// TwinCAT 3 PLC project RoboConnect_Tests
// Title: RoboConnect.Tests
// Company: RoboConnect
// Author: RoboConnect_Maintainer
// ProjectVersion: 0.0.5.0
// Description: 0.1.0.0 Branding update 0.0.5.0 cleans up project 0.0.0.4 updates to new tcrobot 0.0.0.3 Remove tcrobot instances from tests 0.0.0.2 Adds IO tests 0.0.0.1 Adds connection tests
// ProgramVersion: 3.1.4024.0
// libraries:
//   Intecre.Utilities, * (Intecre Ltd)
//   RoboConnect, * (RoboConnect)
//   Tc2_Standard, * (Beckhoff Automation GmbH)
//   tcl_SimpleUnitTestLibrary, * (Red Rock Controls Limited)
// project tree:
//   Code/Mocks/ T_MockBoolCommandTask.TcPOU, T_MockCommandTask.TcPOU, T_MockNumberCommandTask.TcPOU, T_MockTcRobot.TcPOU
//   Code/RoboConnect/Admin Tests/Disable/ T_RoboConnect_Disable_DisabledTrue.TcPOU
//   Code/RoboConnect/Admin Tests/Enable/ T_RoboConnect_Enable_RobotEnabled.TcPOU
//   Code/RoboConnect/ConnectionTests/ T_RoboConnect_WhenCalledWithLowTimeout_FailsConnection.TcPOU, T_RoboConnect_WhenCalled_IsConnectedTrue.TcPOU
//   Code/RoboConnect/IO Tests/AnalogOutput/ T_TcRobot_GetAnalogOutput_CorrectIndexPasses.TcPOU, T_TcRobot_SetAnalogOutput_IncorrectIndexFails.TcPOU, T_TcRobot_SetAnalogOutput_CorrectIndexPasses.TcPOU, T_TcRobot_GetAnalogOutput_IncorrectIndexFails.TcPOU, T_TcRobot_SetAnalogOutput_TimeoutFails.TcPOU
//   Code/RoboConnect/IO Tests/DigitalOutput/ T_TcRobot_SetDigitalOutputTimeout_Fails.TcPOU, T_TcRobot_GetDigitalOutput_CorrectIndexPasses.TcPOU, T_TcRobot_SetDigitalOutput_IncorrectIndexFails.TcPOU, T_TcRobot_SetDigitalOutput_CorrectIndexPasses.TcPOU, T_TcRobot_GetDigitalOutput_ReturnsTrueOutput.TcPOU, T_TcRobot_GetDigitalOutput_IncorrectIndexFails.TcPOU
//   Code/RoboConnect/IO Tests/ToolAnalogOutput/ T_TcRobot_GetToolAnalogOutput_CorrectIndexPasses.TcPOU, T_TcRobot_SetToolAnalogOutput_TimeoutFails.TcPOU, T_TcRobot_SetToolAnalogOutput_IncorrectIndexFails.TcPOU, T_TcRobot_SetToolAnalogOutput_CorrectIndexPasses.TcPOU, T_TcRobot_GetToolAnalogOutput_IncorrectIndexFails.TcPOU
//   Code/RoboConnect/IO Tests/ToolDigitalOutput/ T_TcRobot_SetToolDigitalOutputTimeout_Fails.TcPOU, T_TcRobot_GetToolDigitalOutput_CorrectIndexPasses.TcPOU, T_TcRobot_SetToolDigitalOutput_IncorrectIndexFails.TcPOU, T_TcRobot_SetToolDigitalOutput_CorrectIndexPasses.TcPOU, T_TcRobot_GetToolDigitalOutput_IncorrectIndexFails.TcPOU, T_TcRobot_SetToolDigitalOutput_ReturnsTrueOutput.TcPOU
//   Code/RoboConnect/ T_TcRobot_DisableNotConnected_ReturnsFalse.TcPOU, T_TcRobot_MoveJWrongCount_ReturnsFalse.TcPOU
// (motion and I/O tree: see PLC project roboconnect)
// real-time tasks:
//   TASK PlcTask: cycle T#10ms, priority 22, ADS port 350
//   TASK PlcTask1: cycle T#10ms, priority 21, ADS port 351

// ---- Code/Mocks/T_MockBoolCommandTask.TcPOU
FUNCTION_BLOCK T_MockBoolCommandTask IMPLEMENTS I_BoolResultTask
VAR_INPUT
  _Busy, _Done, _Error, _Timeout : BOOL;
  _Result : BOOL;
END_VAR

METHOD Abort
END_METHOD

PROPERTY Available : BOOL
GET
END_GET
END_PROPERTY

PROPERTY Busy : BOOL
GET
Busy := _busy;
END_GET
END_PROPERTY

METHOD CyclicLogic
END_METHOD

PROPERTY Done : BOOL
GET
Done := _Done;
END_GET
END_PROPERTY

PROPERTY Error : BOOL
GET
Error := _Error;
END_GET
END_PROPERTY

PROPERTY ErrorId : STRING
GET
END_GET
END_PROPERTY

METHOD Execute : BOOL
END_METHOD

METHOD Free
END_METHOD

PROPERTY Result : BOOL
GET
Result := _Result;
END_GET
END_PROPERTY

PROPERTY Timeout : BOOL
GET
Timeout := _Timeout;
END_GET
END_PROPERTY

END_FUNCTION_BLOCK

// ---- Code/Mocks/T_MockCommandTask.TcPOU
FUNCTION_BLOCK T_MockCommandTask IMPLEMENTS I_Task
VAR_INPUT
  _Busy, _Done, _Error, _Timeout : BOOL;
  _Result : LREAL;
END_VAR

METHOD Abort
END_METHOD

PROPERTY Available : BOOL
GET
END_GET
END_PROPERTY

PROPERTY Busy : BOOL
GET
Busy := _Busy;
END_GET
END_PROPERTY

METHOD CyclicLogic
END_METHOD

PROPERTY Done : BOOL
GET
Done := _Done;
END_GET
END_PROPERTY

PROPERTY Error : BOOL
GET
Error := _Error;
END_GET
END_PROPERTY

PROPERTY ErrorId : STRING
GET
END_GET
END_PROPERTY

METHOD Execute : BOOL
END_METHOD

METHOD Free
END_METHOD

PROPERTY Timeout : BOOL
GET
Timeout := _Timeout;
END_GET
END_PROPERTY

END_FUNCTION_BLOCK

// ---- Code/Mocks/T_MockNumberCommandTask.TcPOU
FUNCTION_BLOCK T_MockNumberCommandTask IMPLEMENTS I_NumberResultTask
VAR_INPUT
  _Busy, _Done, _Error, _Timeout : BOOL;
  _Result : LREAL;
END_VAR

METHOD Abort
END_METHOD

PROPERTY Available : BOOL
GET
END_GET
END_PROPERTY

PROPERTY Busy : BOOL
GET
Busy := _Busy;
END_GET
END_PROPERTY

METHOD CyclicLogic
END_METHOD

PROPERTY Done : BOOL
GET
Done := _Done;
END_GET
END_PROPERTY

PROPERTY Error : BOOL
GET
Error := _Error;
END_GET
END_PROPERTY

PROPERTY ErrorId : STRING
GET
END_GET
END_PROPERTY

METHOD Execute : BOOL
END_METHOD

METHOD Free
END_METHOD

PROPERTY Result : LREAL
GET
Result := _Result;
END_GET
END_PROPERTY

PROPERTY Timeout : BOOL
GET
Timeout := _Timeout;
END_GET
END_PROPERTY

END_FUNCTION_BLOCK

// ---- Code/Mocks/T_MockTcRobot.TcPOU
FUNCTION_BLOCK T_MockRoboConnect IMPLEMENTS I_RoboConnect
VAR_INPUT
  _error, _isBusy, _isDone, _isEnabled : BOOL;
  _errorId : UINT;
  _axisCount : UINT;
  _position, _toolPosition : ST_CartesianPoint;
END_VAR
VAR
  state, prevState : (INIT,
    IDLE,
    READY,
    ERROR_STATE) := INIT;

  initalised : BOOL;
  connectionTimer : TON;
  tasktimer : TON;
  _connection : I_Connection;
  _commandQueue : I_CommandQueue;
  _commandTask : T_MockCommandTask;
  _boolCommandTask : T_MockBoolCommandTask;
  _numberCommandTask : T_MockNumberCommandTask;

  digitalOutputs : ARRAY[1..DIGITAL_OUTPUT_COUNT] OF BOOL;
  digitalIntputs : ARRAY[1..DIGITAL_INPUT_COUNT] OF BOOL;
  analogOutputs : ARRAY[1..ANALOG_OUTPUT_COUNT] OF LREAL;
  analogIntputs : ARRAY[1..ANALOG_INPUT_COUNT] OF LREAL;

  toolDigitalOutputs : ARRAY[1..TOOL_DIGITAL_OUTPUT] OF BOOL;
  toolDigitalIntputs : ARRAY[1..TOOL_DIGITAL_INPUT] OF BOOL;
  toolAnalogOutputs : ARRAY[1..TOOL_ANALOG_INPUT] OF LREAL;
  toolAnalogIntputs : ARRAY[1..TOOL_ANALOG_OUTPUT] OF LREAL;

  axes : ARRAY[1..AXIS_COUNT] OF LREAL;

END_VAR
VAR CONSTANT
  DIGITAL_OUTPUT_COUNT : UINT := 6;
  DIGITAL_INPUT_COUNT : UINT := 6;
  ANALOG_INPUT_COUNT : UINT := 6;
  ANALOG_OUTPUT_COUNT : UINT := 6;
  TOOL_ANALOG_OUTPUT : UINT := 2;
  TOOL_DIGITAL_OUTPUT : UINT := 2;
  TOOL_ANALOG_INPUT : UINT := 2;
  TOOL_DIGITAL_INPUT : UINT := 2;
  AXIS_COUNT : UINT := 6;

END_VAR

PROPERTY Busy : BOOL
GET
END_GET
END_PROPERTY

PROPERTY CartesianPosition : TcRobot.ST_CartesianPoint
GET
END_GET
END_PROPERTY

METHOD ClearError : BOOL
VAR_OUTPUT
	task	: TcRobot.I_Task;
END_VAR
END_METHOD

METHOD Connect : BOOL
connectionTimer( IN := FALSE );
connectionTimer( IN := TRUE );
END_METHOD

PROPERTY Connected : BOOL
GET
Connected := connectionTimer.Q;
END_GET
END_PROPERTY

METHOD CyclicLogic
connectionTimer();
taskTimer();

IF taskTimer.Q THEN
  _commandTask(_Timeout := TRUE);
END_IF
END_METHOD

METHOD Disable : BOOL
VAR_OUTPUT
  task : I_Task;
END_VAR
VAR
  resultTask : T_CommandTask;
END_VAR
IF NOT connectionTimer.Q THEN
  task := resultTask;
  RETURN;
END_IF
END_METHOD

METHOD Disconnect : BOOL
VAR_OUTPUT
  task : I_Task;
END_VAR
connectionTimer( IN := FALSE );
END_METHOD

PROPERTY Done : BOOL
GET
END_GET
END_PROPERTY

METHOD Enable : BOOL
VAR_OUTPUT
  task : I_Task;
END_VAR
END_METHOD

PROPERTY Enabled : BOOL
GET
END_GET
END_PROPERTY

PROPERTY Error : BOOL
GET
END_GET
END_PROPERTY

PROPERTY ErrorID : LREAL
GET
END_GET
END_PROPERTY

METHOD GetAnalogOutput : BOOL
VAR_INPUT
  Index : UINT;
END_VAR
VAR_OUTPUT
  task : I_NumberResultTask;
END_VAR
IF Index < 1 OR index > ANALOG_OUTPUT_COUNT THEN
  GetAnalogOutput := FALSE;
  RETURN;
END_IF

_commandTask(_Result := analogOutputs[Index]);
task := _numberCommandTask;

GetAnalogOutput := TRUE;
END_METHOD

METHOD GetAxisCurrents : BOOL
VAR_IN_OUT
  Values : ARRAY[*] OF LREAL;
END_VAR
VAR_OUTPUT
  task : I_Task;
END_VAR
END_METHOD

METHOD GetAxisPositions : BOOL
VAR_IN_OUT
  Values : ARRAY[*] OF LREAL;
END_VAR
VAR_OUTPUT
  task : I_Task;
END_VAR
END_METHOD

METHOD GetAxisTemperatures : BOOL
VAR_IN_OUT
  Values : ARRAY[*] OF LREAL;
END_VAR
VAR_OUTPUT
  task : I_Task;
END_VAR
END_METHOD

METHOD GetDigitalOutput : BOOL
VAR_INPUT
    Index : UINT;
END_VAR
VAR_OUTPUT
  task : I_BoolResultTask;
  value : BOOL;
END_VAR
VAR
  cmdTask : T_CommandTask;
END_VAR
IF Index < 1 OR index > DIGITAL_OUTPUT_COUNT THEN
  GetDigitalOutput := FALSE;
  RETURN;
END_IF

_commandTask(_Result := TO_LREAL(digitalOutputs[Index]), _Done := TRUE);
task := _boolCommandTask;

GetDigitalOutput := TRUE;
END_METHOD

METHOD GetJointPositions : BOOL (* false if incompatible array length*)
VAR_IN_OUT
	(* values overwritten with joint positions.*)
	  joints : ARRAY[*] OF LREAL;
END_VAR
END_METHOD

METHOD GetToolAnalogOutput : BOOL
VAR_INPUT
    Index : UINT;
END_VAR
VAR_OUTPUT
  task : I_NumberResultTask;
END_VAR
IF Index < 1 OR index > DIGITAL_OUTPUT_COUNT THEN
  GetToolAnalogOutput := FALSE;
  RETURN;
END_IF

_commandTask(_Result := toolAnalogOutputs[Index]);
task := _numberCommandTask;

GetToolAnalogOutput := TRUE;
END_METHOD

METHOD GetToolDigitalOutput : BOOL
VAR_INPUT
	Index	: UINT;
END_VAR
VAR_OUTPUT
	task	: I_BoolResultTask;
END_VAR
IF Index < 1 OR Index > TOOL_DIGITAL_OUTPUT THEN
  GetToolDigitalOutput := FALSE;
  RETURN;
END_IF

_commandTask(_Result := TO_LREAL(toolDigitalOutputs[Index]));
task := _boolCommandTask;

GetToolDigitalOutput := TRUE;
END_METHOD

METHOD Halt : BOOL
VAR_OUTPUT
  task : I_Task;
END_VAR
END_METHOD

METHOD IsAtCartesianPosition : BOOL
VAR_INPUT
	point	: TcRobot.ST_CartesianPoint;
END_VAR
END_METHOD

METHOD IsAtJointPosition : BOOL
VAR_IN_OUT
	(* positions 1..NumberOfAxes will be used. passed array should be dimensioned accordingly*)
  joints : ARRAY[*] OF LREAL; // positions 1..NumberOfAxes will be used. passed array should be dimensioned accordingly
END_VAR
END_METHOD

METHOD JogAxis : BOOL // default tool and user frame
VAR_INPUT
  axisIndex : UDINT; // joint or enumerated cartesian direction/vector. See concrete type docs for enumeration of cartesian coords.
  axisDirection : BOOL; // TRUE = positive, FALSE = negative
  jogType : E_JogType; // Cartesian or Joint space
END_VAR
VAR_OUTPUT
	task	: TcRobot.I_Task;
END_VAR
END_METHOD

METHOD JogAxisAdvanced : BOOL
VAR_INPUT
  axisIndex : UDINT; // joint or enumerated cartesian direction/vector. See concrete type docs for enumeration of cartesian coords.
  axisDirection : BOOL; // TRUE = positive, FALSE = negative
  jogType : E_JogType; // Cartesian or Joint space
  coordType : INT; // set to 0 to leave default
  user : INT; // set to 0 to leave default
  tool : INT; // set to 0 to leave default
END_VAR
VAR_OUTPUT
	task	: TcRobot.I_Task;
END_VAR
END_METHOD

PROPERTY Manufacturer : STRING
GET
END_GET
END_PROPERTY

PROPERTY Model : STRING
GET
END_GET
END_PROPERTY

METHOD MoveAbs : BOOL
VAR_INPUT
  point : ST_CartesianPoint;
END_VAR
VAR_OUTPUT
  task : I_Task;
END_VAR
END_METHOD

METHOD MoveJ : BOOL
VAR_IN_OUT
  joints : ARRAY[*] OF LREAL;
END_VAR
VAR_OUTPUT
  task : I_Task;
END_VAR
VAR
  returnedTask : T_CommandTask;
END_VAR
IF UPPER_BOUND(joints,1) > _axisCount THEN
  task := returnedTask;
  RETURN;
END_IF
END_METHOD

PROPERTY Position : ST_CartesianPoint
GET
END_GET
END_PROPERTY

METHOD Reset : BOOL
VAR_OUTPUT
  task : I_Task;
END_VAR
END_METHOD

PROPERTY Running : BOOL
GET
END_GET
END_PROPERTY

METHOD SetAnalogOutput : BOOL
VAR_INPUT
  Index : UINT;
  Value : LREAL;
END_VAR
VAR_OUTPUT
  task : I_Task;
END_VAR
IF Index < 1 OR index > DIGITAL_OUTPUT_COUNT THEN
  SetAnalogOutput := FALSE;
  RETURN;
END_IF

tasktimer.IN := FALSE;
tasktimer.IN := TRUE;

analogOutputs[Index] := Value;
task := _commandTask;

SetAnalogOutput := TRUE;
END_METHOD

METHOD SetAtPosDeltas : BOOL
VAR_INPUT
  atPosCartesianDeltas : ST_CartesianPoint;
END_VAR
VAR_IN_OUT
  atPosJointDeltas : ARRAY[*] OF LREAL; // positions 1..NumberOfAxes will be used. passed array should be dimensioned accordingly
END_VAR
END_METHOD

METHOD SetBufferMode : BOOL
VAR_INPUT
  BufferMode : E_BufferMode;
END_VAR
END_METHOD

METHOD SetCarteasianAcceleration : BOOL
VAR_INPUT
  Acceleration : LREAL;
END_VAR
VAR_OUTPUT
  task : I_Task;
END_VAR
END_METHOD

METHOD SetCartesianSpeed : BOOL
VAR_INPUT
  Speed : LREAL;
END_VAR
VAR_OUTPUT
  task : I_Task;
END_VAR
END_METHOD

METHOD PUBLIC SetConnectionTime  // set simulated connection time
VAR_INPUT
  connectionTime : TIME;
END_VAR
connectionTimer.PT := connectionTime;
END_METHOD

METHOD SetDigitalOutput : BOOL
VAR_INPUT
  Index : UINT;
  Value : BOOL;
END_VAR
VAR_OUTPUT
  task : I_Task;
END_VAR
IF Index < 1 OR index > DIGITAL_OUTPUT_COUNT THEN
  SetDigitalOutput := FALSE;
  RETURN;
END_IF

tasktimer.IN := FALSE;
tasktimer.IN := TRUE;

digitalOutputs[Index] := TRUE;
_commandTask(_Done := TRUE);
task := _commandTask;

SetDigitalOutput := TRUE;
END_METHOD

METHOD PUBLIC SetGeneralCommandResponseDuration : BOOL // This sets the duration that the task will take, used for causing timeout or done in the returned task
VAR_INPUT
    taskTime : TIME;
END_VAR
tasktimer.PT := taskTime;
END_METHOD

METHOD SetJogType : BOOL
VAR_INPUT
  JogType : E_JogType;
END_VAR
VAR_OUTPUT
  task : I_Task;
END_VAR
END_METHOD

METHOD SetJointAcceleration : BOOL
VAR_INPUT
  Acceleration : LREAL;
END_VAR
VAR_OUTPUT
  task : I_Task;
END_VAR
END_METHOD

METHOD SetJointSpeed : BOOL
VAR_INPUT
  Speed : LREAL;
END_VAR
VAR_OUTPUT
  task : I_Task;
END_VAR
END_METHOD

METHOD SetToolAnalogOutput : BOOL
VAR_INPUT
  Index : UINT;
  Value : LREAL;
END_VAR
VAR_OUTPUT
  task : I_Task;
END_VAR
IF Index > ANALOG_OUTPUT_COUNT THEN
  SetToolAnalogOutput := FALSE;
  RETURN;
END_IF

tasktimer.IN := FALSE;
tasktimer.IN := TRUE;

toolDigitalOutputs[Index] := TRUE;
task := _commandTask;

SetToolAnalogOutput := TRUE;
END_METHOD

METHOD SetToolDigitalOutput : BOOL
VAR_INPUT
	Index	: UINT;
	Value	: BOOL;
END_VAR
VAR_OUTPUT
	task	: TcRobot.I_Task;
END_VAR
IF Index < 1 OR Index > TOOL_ANALOG_OUTPUT THEN
  SetToolDigitalOutput := FALSE;
  RETURN;
END_IF

tasktimer.IN := FALSE;
tasktimer.IN := TRUE;

toolDigitalOutputs[Index] := TRUE;
task := _commandTask;

SetToolDigitalOutput := TRUE;
END_METHOD

METHOD SetToolFrame : BOOL
VAR_INPUT
 Frame : ST_CartesianPoint;
END_VAR
VAR_OUTPUT
  task : I_Task;
END_VAR
END_METHOD

METHOD SetTransitionMode : BOOL
VAR_INPUT
END_VAR
END_METHOD

METHOD SetTransitionParameter : BOOL
VAR_INPUT
  CPratio : LREAL;
END_VAR
VAR_OUTPUT
	task	: TcRobot.I_Task;
END_VAR
END_METHOD

METHOD SetUserFrame : BOOL
VAR_INPUT
  Frame : ST_CartesianPoint;
END_VAR
VAR_OUTPUT
	task : I_Task;
END_VAR
END_METHOD

METHOD Stop : BOOL
VAR_OUTPUT
  task : I_Task;
END_VAR
END_METHOD

PROPERTY ToolPosition : ST_CartesianPoint
GET
END_GET
END_PROPERTY

END_FUNCTION_BLOCK

// ---- Code/RoboConnect/Admin Tests/Disable/T_RoboConnect_Disable_DisabledTrue.TcPOU
FUNCTION_BLOCK T_RoboConnect_Disable_DisabledTrue EXTENDS T_UnitTestBase
VAR
  _robot : I_RoboConnect;
  myTestState, prevState : (ARRANGE, ACT, ASSERT);
  actual : STRING;
  expected : STRING := '0';
  resultTask : I_Task;
END_VAR

CASE myTestState OF
  ARRANGE:
    StateChanged();
    myTestState := ACT;

  ACT:
  IF StateChanged() THEN
    _robot.Enable(task => resultTask);
    
	ELSIF NOT resultTask.Busy THEN
        myTestState := ASSERT;
  END_IF
  
  ASSERT:
    actual := resultTask.ErrorId;
    assertion.AssertEquals_STRING(expected, actual, 'actual := _robot.Enabled;');
    myTestState := ARRANGE;
    TestFinished();
END_CASE

METHOD FB_init : BOOL
VAR_INPUT
  bInitRetains : BOOL; // if TRUE, the retain variables are initialized (warm start / cold start)
  bInCopyCode : BOOL; // if TRUE, the instance afterwards gets moved into the copy code (online change)
  TestSuite : I_TestSuite;
  robot : I_TcRobot;
END_VAR
_robot := robot;
END_METHOD

METHOD PRIVATE StateChanged : BOOL
IF  myTestState = prevState THEN
  RETURN;
END_IF

prevState := myTestState;
StateChanged := TRUE;
END_METHOD

METHOD WaitForCycles : BOOL
VAR_INPUT
  maxCount : UINT;
END_VAR
counter := counter + 1;

IF counter = maxCount THEN
  counter := 0;
  WaitForCycles := TRUE;
END_IF
END_METHOD

END_FUNCTION_BLOCK

// ---- Code/RoboConnect/Admin Tests/Enable/T_RoboConnect_Enable_RobotEnabled.TcPOU
FUNCTION_BLOCK T_RoboConnect_Enable_RobotEnabled EXTENDS T_UnitTestBase
VAR
  _robot : I_RoboConnect;
  myTestState, prevState : (ARRANGE, ACT, ASSERT);
  actual : STRING;
  expected : STRING := '0';
  resultTask : I_Task;
END_VAR

CASE myTestState OF
  ARRANGE:
    StateChanged();
    myTestState := ACT;

  ACT:
  IF StateChanged() THEN
    _robot.Enable(task => resultTask);
    
	ELSIF NOT resultTask.Busy THEN
        myTestState := ASSERT;
  END_IF
  
  ASSERT:
    actual := resultTask.ErrorId;
    assertion.AssertEquals_STRING(expected, actual, 'actual := _robot.Enabled;');
    myTestState := ARRANGE;
    TestFinished();
END_CASE

METHOD FB_init : BOOL
VAR_INPUT
  bInitRetains : BOOL; // if TRUE, the retain variables are initialized (warm start / cold start)
  bInCopyCode : BOOL; // if TRUE, the instance afterwards gets moved into the copy code (online change)
  TestSuite : I_TestSuite;
  robot : I_TcRobot;
END_VAR
_robot := robot;
END_METHOD

METHOD PRIVATE StateChanged : BOOL
IF  myTestState = prevState THEN
  RETURN;
END_IF

prevState := myTestState;
StateChanged := TRUE;
END_METHOD

METHOD WaitForCycles : BOOL
VAR_INPUT
  maxCount : UINT;
END_VAR
counter := counter + 1;

IF counter = maxCount THEN
  counter := 0;
  WaitForCycles := TRUE;
END_IF
END_METHOD

END_FUNCTION_BLOCK

// ---- Code/RoboConnect/ConnectionTests/T_RoboConnect_WhenCalledWithLowTimeout_FailsConnection.TcPOU
FUNCTION_BLOCK T_RoboConnect_WhenCalledWithLowTimeout_FailsConnection EXTENDS T_UnitTestBase
VAR
  robot : I_RoboConnect;
  timeOutTimer : TON;
  myTestState, prevState : (INIT, ARRANGE, ACT, ASSERT) := INIT;
  expected, actual : BOOL;
  counter : UINT;
END_VAR

CASE myTestState OF
  INIT:
    StateChanged();
    myTestState := ARRANGE;

  ARRANGE:
    StateChanged();

    expected := FALSE;
    myTestState := ACT;

  ACT:
    robot.Connect();
    myTestState := ASSERT;

  ASSERT:

    IF timeOutTimer.Q THEN
      actual := robot.Connected;
      assertion.AssertEquals_BOOL(expected, actual, 'IsConnected := FALSE');
      TestFinished();
      myTestState := INIT;
      robot.Disconnect();
    END_IF

END_CASE

timeOutTimer(IN := myTestState = ASSERT);

METHOD FB_init : BOOL
VAR_INPUT
  bInitRetains : BOOL; // if TRUE, the retain variables are initialized (warm start / cold start)
  bInCopyCode : BOOL; // if TRUE, the instance afterwards gets moved into the copy code (online change)
  TestSuite : tcl_SimpleUnitTestLibrary.I_TestSuite;
  robot : I_TcRobot;
  timeout : TIME;
END_VAR
THIS^.robot := robot;
THIS^.timeOutTimer.PT := timeout;
END_METHOD

METHOD PRIVATE StateChanged : BOOL
IF  myTestState = prevState THEN
  RETURN;
END_IF

prevState := myTestState;
StateChanged := TRUE;
END_METHOD

METHOD WaitForCycles : BOOL
VAR_INPUT
  maxCount : UINT;
END_VAR
counter := counter + 1;

IF counter = maxCount THEN
  counter := 0;
  WaitForCycles := TRUE;
END_IF
END_METHOD

END_FUNCTION_BLOCK

// ---- Code/RoboConnect/ConnectionTests/T_RoboConnect_WhenCalled_IsConnectedTrue.TcPOU
FUNCTION_BLOCK T_RoboConnect_WhenCalled_IsConnectedTrue EXTENDS T_UnitTestBase
VAR
  robot : I_RoboConnect;
  timeOutTimer : TON;
  myTestState, prevState : (INIT, ARRANGE, ACT, ASSERT) := INIT;
  expected, actual : BOOL;
  counter : UINT;
END_VAR

CASE myTestState OF
  INIT:
    StateChanged();
    myTestState := ARRANGE;

  ARRANGE:
    StateChanged();

    expected := TRUE;
    myTestState := ACT;

  ACT:
    robot.Connect();
    myTestState := ASSERT;

  ASSERT:

    IF robot.Connected OR timeOutTimer.Q THEN
      actual := robot.Connected;
      assertion.AssertEquals_BOOL(expected, actual, 'IsConnected := TRUE');
      TestFinished();
      myTestState := INIT;
      // dont disconnect here, connection is required for the next test
    END_IF

END_CASE

timeOutTimer(IN := myTestState = ASSERT);

METHOD FB_init : BOOL
VAR_INPUT
  bInitRetains : BOOL; // if TRUE, the retain variables are initialized (warm start / cold start)
  bInCopyCode : BOOL; // if TRUE, the instance afterwards gets moved into the copy code (online change)
  TestSuite : tcl_SimpleUnitTestLibrary.I_TestSuite;
  robot : I_TcRobot;
  timeout : TIME;
END_VAR
THIS^.robot := robot;
THIS^.timeOutTimer.PT := timeout;
END_METHOD

METHOD PRIVATE StateChanged : BOOL
IF  myTestState = prevState THEN
  RETURN;
END_IF

prevState := myTestState;
StateChanged := TRUE;
END_METHOD

METHOD WaitForCycles : BOOL
VAR_INPUT
  maxCount : UINT;
END_VAR
counter := counter + 1;

IF counter = maxCount THEN
  counter := 0;
  WaitForCycles := TRUE;
END_IF
END_METHOD

END_FUNCTION_BLOCK

// ---- Code/RoboConnect/IO Tests/AnalogOutput/T_TcRobot_GetAnalogOutput_CorrectIndexPasses.TcPOU
FUNCTION_BLOCK T_RoboConnect_GetAnalogOutput_CorrectIndexPasses EXTENDS T_UnitTestBase
VAR
  robot : I_RoboConnect;
  targetDO : UINT;
  myTestState, prevState :
    (INIT, ARRANGE, ACT, ASSERT) := INIT;
  expected, actual : BOOL;
  counter : UINT;
  returnedTask : I_Task;
  resultTask : I_NumberResultTask;
END_VAR

CASE myTestState OF
  INIT:
    StateChanged();
    myTestState := ARRANGE;

  ARRANGE:
    IF StateChanged() THEN
      expected := TRUE;
      myTestState := ACT;
    END_IF

  ACT:
    actual := robot.GetAnalogOutput(targetDO, task => resultTask);
    myTestState := ASSERT;

  ASSERT:
    assertion.AssertEquals_BOOL(expected, actual, 'robot.GetAnalogOutput(targetDO, task => returnedTask)');
    TestFinished();
    myTestState := INIT;

END_CASE

METHOD FB_init : BOOL
VAR_INPUT
  bInitRetains : BOOL; // if TRUE, the retain variables are initialized (warm start / cold start)
  bInCopyCode : BOOL; // if TRUE, the instance afterwards gets moved into the copy code (online change)
  TestSuite : tcl_SimpleUnitTestLibrary.I_TestSuite;
  robot : I_TcRobot;
  targetDo : UINT;
END_VAR
THIS^.robot := robot;
THIS^.targetDo := targetDo;
END_METHOD

METHOD PRIVATE StateChanged : BOOL
IF  myTestState = prevState THEN
  RETURN;
END_IF

prevState := myTestState;
StateChanged := TRUE;
END_METHOD

METHOD WaitForCycles : BOOL
VAR_INPUT
  maxCount : UINT;
END_VAR
counter := counter + 1;

IF counter = maxCount THEN
  counter := 0;
  WaitForCycles := TRUE;
END_IF
END_METHOD

END_FUNCTION_BLOCK

// ---- Code/RoboConnect/IO Tests/AnalogOutput/T_TcRobot_SetAnalogOutput_IncorrectIndexFails.TcPOU
FUNCTION_BLOCK T_RoboConnect_SetAnalogOutput_IncorrectIndexFails EXTENDS T_UnitTestBase
VAR
  robot : I_RoboConnect;
  targetDO : UINT;
  myTestState, prevState :
    (INIT, ARRANGE, ACT, ASSERT) := INIT;
  expected: BOOL;
  actual : BOOL := TRUE;
  counter : UINT;
END_VAR

CASE myTestState OF
  INIT:
    StateChanged();
    myTestState := ARRANGE;

  ARRANGE:
    IF StateChanged() THEN
      expected := FALSE;
      myTestState := ACT;
    END_IF

  ACT:
    actual := robot.SetAnalogOutput(targetDO, 0.5);
    myTestState := ASSERT;

  ASSERT:
    assertion.AssertEquals_BOOL(expected, actual, 'robot.SetAnalogOutput(targetDO,TRUE)');
    TestFinished();
    myTestState := INIT;

END_CASE

METHOD FB_init : BOOL
VAR_INPUT
  bInitRetains : BOOL; // if TRUE, the retain variables are initialized (warm start / cold start)
  bInCopyCode : BOOL; // if TRUE, the instance afterwards gets moved into the copy code (online change)
  TestSuite : tcl_SimpleUnitTestLibrary.I_TestSuite;
  robot : I_TcRobot;
  targetDo : UINT;
END_VAR
THIS^.robot := robot;
THIS^.targetDo := targetDo;
END_METHOD

METHOD PRIVATE StateChanged : BOOL
IF  myTestState = prevState THEN
  RETURN;
END_IF

prevState := myTestState;
StateChanged := TRUE;
END_METHOD

METHOD WaitForCycles : BOOL
VAR_INPUT
  maxCount : UINT;
END_VAR
counter := counter + 1;

IF counter = maxCount THEN
  counter := 0;
  WaitForCycles := TRUE;
END_IF
END_METHOD

END_FUNCTION_BLOCK

// ---- Code/RoboConnect/IO Tests/AnalogOutput/T_TcRobot_SetAnalogOutput_CorrectIndexPasses.TcPOU
FUNCTION_BLOCK T_RoboConnect_SetAnalogOutput_CorrectIndexPasses EXTENDS T_UnitTestBase
VAR
  robot : I_RoboConnect;
  targetDO : UINT;
  myTestState, prevState :
    (INIT, ARRANGE, ACT, ASSERT) := INIT;
  expected, actual : BOOL;
  counter : UINT;
END_VAR

CASE myTestState OF
  INIT:
    StateChanged();
    myTestState := ARRANGE;

  ARRANGE:
    IF StateChanged() THEN
      expected := TRUE;
      myTestSTate := ACT;
    END_IF

  ACT:
    actual := robot.SetAnalogOutput(targetDO, 0.5);
    myTestState := ASSERT;

  ASSERT:
    assertion.AssertEquals_BOOL(expected, actual, 'robot.SetAnalogOutput(targetDO,TRUE)');
    TestFinished();
    myTestState := INIT;

END_CASE

METHOD FB_init : BOOL
VAR_INPUT
  bInitRetains : BOOL; // if TRUE, the retain variables are initialized (warm start / cold start)
  bInCopyCode : BOOL; // if TRUE, the instance afterwards gets moved into the copy code (online change)
  TestSuite : tcl_SimpleUnitTestLibrary.I_TestSuite;
  robot : I_TcRobot;
  targetDo : UINT;
END_VAR
THIS^.robot := robot;
THIS^.targetDo := targetDo;
END_METHOD

METHOD PRIVATE StateChanged : BOOL
IF  myTestState = prevState THEN
  RETURN;
END_IF

prevState := myTestState;
StateChanged := TRUE;
END_METHOD

METHOD WaitForCycles : BOOL
VAR_INPUT
  maxCount : UINT;
END_VAR
counter := counter + 1;

IF counter = maxCount THEN
  counter := 0;
  WaitForCycles := TRUE;
END_IF
END_METHOD

END_FUNCTION_BLOCK

// ---- Code/RoboConnect/IO Tests/AnalogOutput/T_TcRobot_GetAnalogOutput_IncorrectIndexFails.TcPOU
FUNCTION_BLOCK T_RoboConnect_GetAnalogOutput_IncorrectIndexFails EXTENDS T_UnitTestBase
VAR
  robot : I_RoboConnect;
  targetDO : UINT;
  myTestState, prevState :
    (INIT, ARRANGE, ACT, ASSERT) := INIT;
  expected : BOOL;
  actual : BOOL := TRUE;
  counter : UINT;
  returnedTask : I_Task;
  resultTask : I_NumberResultTask;
END_VAR

CASE myTestState OF
  INIT:
    StateChanged();
    myTestState := ARRANGE;

  ARRANGE:
    IF StateChanged() THEN
      expected := FALSE;
      myTestState := ACT;
    END_IF

  ACT:
    actual := robot.GetAnalogOutput(targetDO, task => resultTask);
    myTestState := ASSERT;

  ASSERT:
    assertion.AssertEquals_BOOL(expected, actual, 'returnedTask');
    TestFinished();
    myTestState := INIT;

END_CASE

METHOD FB_init : BOOL
VAR_INPUT
  bInitRetains : BOOL; // if TRUE, the retain variables are initialized (warm start / cold start)
  bInCopyCode : BOOL; // if TRUE, the instance afterwards gets moved into the copy code (online change)
  TestSuite : tcl_SimpleUnitTestLibrary.I_TestSuite;
  robot : I_TcRobot;
  targetDo : UINT;
END_VAR
THIS^.robot := robot;
THIS^.targetDo := targetDo;
END_METHOD

METHOD PRIVATE StateChanged : BOOL
IF  myTestState = prevState THEN
  RETURN;
END_IF

prevState := myTestState;
StateChanged := TRUE;
END_METHOD

METHOD WaitForCycles : BOOL
VAR_INPUT
  maxCount : UINT;
END_VAR
counter := counter + 1;

IF counter = maxCount THEN
  counter := 0;
  WaitForCycles := TRUE;
END_IF
END_METHOD

END_FUNCTION_BLOCK

// ---- Code/RoboConnect/IO Tests/AnalogOutput/T_TcRobot_SetAnalogOutput_TimeoutFails.TcPOU
FUNCTION_BLOCK T_RoboConnect_SetAnalogOutput_TimeoutFails EXTENDS T_UnitTestBase
VAR
  robot : I_RoboConnect;
  timeOutTimer : TON;
  targetAO : UINT;
  myTestState, prevState :
    (INIT,
    ARRANGE,
    ACT,
    ASSERT) := INIT;
  expected, actual : BOOL;
  counter : UINT;
  returnedTask : I_Task;
END_VAR

CASE myTestState OF
  INIT:
    StateChanged();
    myTestState := ARRANGE;

  ARRANGE:
    IF StateChanged() THEN
      expected := TRUE;
      robot.Connect();
    END_IF

    IF robot.Connected THEN
      myTestState := ACT;
    END_IF

  ACT:
    robot.SetDigitalOutput(targetAO,TRUE, task => returnedTask);
    myTestState := ASSERT;

  ASSERT:
    IF timeOutTimer.Q THEN
      actual := returnedTask.Timeout;
      assertion.AssertEquals_BOOL(expected, actual, 'actual := returnedTask.Timeout');
      TestFinished();
      myTestState := INIT;

    END_IF

END_CASE

robot.CyclicLogic();
timeOutTimer(IN := myTestState = ASSERT);

METHOD FB_init : BOOL
VAR_INPUT
  bInitRetains : BOOL; // if TRUE, the retain variables are initialized (warm start / cold start)
  bInCopyCode : BOOL; // if TRUE, the instance afterwards gets moved into the copy code (online change)
  TestSuite : tcl_SimpleUnitTestLibrary.I_TestSuite;
  robot : I_TcRobot;
  targetAo : UINT;
  timeout : TIME;
END_VAR
THIS^.robot := robot;
THIS^.timeoutTimer.PT := timeout;
THIS^.targetAo := targetAo;
END_METHOD

METHOD PRIVATE StateChanged : BOOL
IF  myTestState = prevState THEN
  RETURN;
END_IF

prevState := myTestState;
StateChanged := TRUE;
END_METHOD

METHOD WaitForCycles : BOOL
VAR_INPUT
  maxCount : UINT;
END_VAR
counter := counter + 1;

IF counter = maxCount THEN
  counter := 0;
  WaitForCycles := TRUE;
END_IF
END_METHOD

END_FUNCTION_BLOCK

// ---- Code/RoboConnect/IO Tests/DigitalOutput/T_TcRobot_SetDigitalOutputTimeout_Fails.TcPOU
FUNCTION_BLOCK T_RoboConnect_SetDigitalOutputTimeout_Fails EXTENDS T_UnitTestBase
VAR
  robot : I_RoboConnect;
  timeOutTimer : TON;
  targetDO : UINT;
  myTestState, prevState :
    (INIT, ARRANGE, ACT, ASSERT) := INIT;
  expected, actual : BOOL;
  counter : UINT;
  returnedTask : I_Task;
END_VAR

CASE myTestState OF
  INIT:
    StateChanged();
    myTestState := ARRANGE;

  ARRANGE:
    IF StateChanged() THEN
      expected := TRUE;
      robot.Connect();
    END_IF

    IF robot.Connected THEN
      myTestState := ACT;
    END_IF

  ACT:
    robot.SetDigitalOutput(targetDO,TRUE, task => returnedTask);
    myTestState := ASSERT;

  ASSERT:
    IF timeOutTimer.Q THEN
      actual := returnedTask.Timeout;
      assertion.AssertEquals_BOOL(expected, actual, 'actual := returnedTask.Timeout');
      TestFinished();
      myTestState := INIT;

    END_IF

END_CASE

robot.CyclicLogic();
timeOutTimer(IN := myTestState = ASSERT);

METHOD FB_init : BOOL
VAR_INPUT
  bInitRetains : BOOL; // if TRUE, the retain variables are initialized (warm start / cold start)
  bInCopyCode : BOOL; // if TRUE, the instance afterwards gets moved into the copy code (online change)
  TestSuite : tcl_SimpleUnitTestLibrary.I_TestSuite;
  robot : I_TcRobot;
  targetDo : UINT;
  timeout : TIME;
END_VAR
THIS^.robot := robot;
THIS^.timeoutTimer.PT := timeout;
THIS^.targetDo := targetDo;
END_METHOD

METHOD PRIVATE StateChanged : BOOL
IF  myTestState = prevState THEN
  RETURN;
END_IF

prevState := myTestState;
StateChanged := TRUE;
END_METHOD

METHOD WaitForCycles : BOOL
VAR_INPUT
  maxCount : UINT;
END_VAR
counter := counter + 1;

IF counter = maxCount THEN
  counter := 0;
  WaitForCycles := TRUE;
END_IF
END_METHOD

END_FUNCTION_BLOCK

// ---- Code/RoboConnect/IO Tests/DigitalOutput/T_TcRobot_GetDigitalOutput_CorrectIndexPasses.TcPOU
FUNCTION_BLOCK T_RoboConnect_GetDigitalOutput_CorrectIndexPasses EXTENDS T_UnitTestBase
VAR
  robot : I_RoboConnect;
  targetDO : UINT;
  myTestState, prevState :
    (INIT, ARRANGE, ACT, ASSERT) := INIT;
  expected, actual : BOOL;
  counter : UINT;
  returnedTask : I_Task;
  resultTask : I_BoolResultTask;
END_VAR

CASE myTestState OF
  INIT:
    StateChanged();
    myTestState := ARRANGE;

  ARRANGE:
    IF StateChanged() THEN
      expected := TRUE;
      myTestState := ACT;
    END_IF

  ACT:
    actual := robot.GetDigitalOutput(targetDO, task => resultTask);
    myTestState := ASSERT;

  ASSERT:
    assertion.AssertEquals_BOOL(expected, actual, 'robot.GetDigitalOutput(targetDO, task => returnedTask)');
    TestFinished();
    myTestState := INIT;

END_CASE

METHOD FB_init : BOOL
VAR_INPUT
  bInitRetains : BOOL; // if TRUE, the retain variables are initialized (warm start / cold start)
  bInCopyCode : BOOL; // if TRUE, the instance afterwards gets moved into the copy code (online change)
  TestSuite : tcl_SimpleUnitTestLibrary.I_TestSuite;
  robot : I_TcRobot;
  targetDo : UINT;
END_VAR
THIS^.robot := robot;
THIS^.targetDo := targetDo;
END_METHOD

METHOD PRIVATE StateChanged : BOOL
IF  myTestState = prevState THEN
  RETURN;
END_IF

prevState := myTestState;
StateChanged := TRUE;
END_METHOD

METHOD WaitForCycles : BOOL
VAR_INPUT
  maxCount : UINT;
END_VAR
counter := counter + 1;

IF counter = maxCount THEN
  counter := 0;
  WaitForCycles := TRUE;
END_IF
END_METHOD

END_FUNCTION_BLOCK

// ---- Code/RoboConnect/IO Tests/DigitalOutput/T_TcRobot_SetDigitalOutput_IncorrectIndexFails.TcPOU
FUNCTION_BLOCK T_RoboConnect_SetDigitalOutput_IncorrectIndexFails EXTENDS T_UnitTestBase
VAR
  robot : I_RoboConnect;
  targetDO : UINT;
  myTestState, prevState :
    (INIT, ARRANGE, ACT, ASSERT) := INIT;
  expected : BOOL;
  actual : BOOL := TRUE;
  counter : UINT;
END_VAR

CASE myTestState OF
  INIT:
    StateChanged();
    myTestState := ARRANGE;

  ARRANGE:
    IF StateChanged() THEN
      expected := FALSE;
      myTestState := ACT;
    END_IF

  ACT:
    actual := robot.SetDigitalOutput(targetDO, TRUE);
    myTestState := ASSERT;

  ASSERT:
    actual := robot.GetDigitalOutput(targetDO);
    assertion.AssertEquals_BOOL(expected, actual, 'actual := robot.SetDigitalOutput(targetDO, TRUE)');
    TestFinished();
    myTestState := INIT;

END_CASE

METHOD FB_init : BOOL
VAR_INPUT
  bInitRetains : BOOL; // if TRUE, the retain variables are initialized (warm start / cold start)
  bInCopyCode : BOOL; // if TRUE, the instance afterwards gets moved into the copy code (online change)
  TestSuite : tcl_SimpleUnitTestLibrary.I_TestSuite;
  robot : I_TcRobot;
  targetDo : UINT;
END_VAR
THIS^.robot := robot;
THIS^.targetDo := targetDo;
END_METHOD

METHOD PRIVATE StateChanged : BOOL
IF  myTestState = prevState THEN
  RETURN;
END_IF

prevState := myTestState;
StateChanged := TRUE;
END_METHOD

METHOD WaitForCycles : BOOL
VAR_INPUT
  maxCount : UINT;
END_VAR
counter := counter + 1;

IF counter = maxCount THEN
  counter := 0;
  WaitForCycles := TRUE;
END_IF
END_METHOD

END_FUNCTION_BLOCK

// ---- Code/RoboConnect/IO Tests/DigitalOutput/T_TcRobot_SetDigitalOutput_CorrectIndexPasses.TcPOU
FUNCTION_BLOCK T_RoboConnect_SetDigitalOutput_CorrectIndexPasses EXTENDS T_UnitTestBase
VAR
  robot : I_RoboConnect;
  targetDO : UINT;
  myTestState, prevState :
    (INIT, ARRANGE, ACT, ASSERT) := INIT;
  expected, actual : BOOL;
  counter : UINT;
END_VAR

CASE myTestState OF
  INIT:
    StateChanged();
    myTestState := ARRANGE;

  ARRANGE:
    IF StateChanged() THEN
      expected := TRUE;
      robot.Connect();
    END_IF

    IF robot.Connected THEN
      myTestState := ACT;
    END_IF

  ACT:
    actual := robot.SetDigitalOutput(targetDO, TRUE);
    myTestState := ASSERT;

  ASSERT:
    actual := robot.GetDigitalOutput(targetDO);
    assertion.AssertEquals_BOOL(expected, actual, 'actual := robot.SetDigitalOutput(targetDO, TRUE)');
    TestFinished();
    myTestState := INIT;

END_CASE

METHOD FB_init : BOOL
VAR_INPUT
  bInitRetains : BOOL; // if TRUE, the retain variables are initialized (warm start / cold start)
  bInCopyCode : BOOL; // if TRUE, the instance afterwards gets moved into the copy code (online change)
  TestSuite : tcl_SimpleUnitTestLibrary.I_TestSuite;
  robot : I_TcRobot;
  targetDo : UINT;
END_VAR
THIS^.robot := robot;
THIS^.targetDo := targetDo;
END_METHOD

METHOD PRIVATE StateChanged : BOOL
IF  myTestState = prevState THEN
  RETURN;
END_IF

prevState := myTestState;
StateChanged := TRUE;
END_METHOD

METHOD WaitForCycles : BOOL
VAR_INPUT
  maxCount : UINT;
END_VAR
counter := counter + 1;

IF counter = maxCount THEN
  counter := 0;
  WaitForCycles := TRUE;
END_IF
END_METHOD

END_FUNCTION_BLOCK

// ---- Code/RoboConnect/IO Tests/DigitalOutput/T_TcRobot_GetDigitalOutput_ReturnsTrueOutput.TcPOU
FUNCTION_BLOCK T_RoboConnect_GetDigitalOutput_ReturnsTrueOutput EXTENDS T_UnitTestBase
VAR
  robot : I_RoboConnect;
  timeOutTimer : TON;
  targetDO : UINT;
  targetDoState : BOOL;
  myTestState, prevState :
    (INIT, ARRANGE, ACT, ASSERT) := INIT;
  expected, actual : BOOL;
  counter : UINT;
  returnedTask : I_Task;
  boolResultTask : I_BoolResultTask;
END_VAR

CASE myTestState OF
  INIT:
    StateChanged();
    myTestState := ARRANGE;

  ARRANGE:
    IF StateChanged() THEN
      expected := targetDoState;
      robot.SetDigitalOutput(targetDO, targetDoState, task => returnedTask);
    END_IF

    IF returnedTask.Done THEN
      myTestState := ACT;
    END_IF

  ACT:
    IF StateChanged() THEN
      robot.GetDigitalOutput(targetDO, task => boolResultTask);
    END_IF

    myTestState := ASSERT;

  ASSERT:
    actual := boolResultTask.Result;
    assertion.AssertEquals_BOOL(expected, actual, 'robot.GetDigitalOutput(targetDO) := TRUE');
    TestFinished();
    myTestState := INIT;

END_CASE

robot.CyclicLogic();
timeOutTimer(IN := myTestState = ASSERT);

METHOD FB_init : BOOL
VAR_INPUT
  bInitRetains : BOOL; // if TRUE, the retain variables are initialized (warm start / cold start)
  bInCopyCode : BOOL; // if TRUE, the instance afterwards gets moved into the copy code (online change)
  TestSuite : tcl_SimpleUnitTestLibrary.I_TestSuite;
  robot : I_TcRobot;
  targetDo : UINT; // the output enumeration
  targetDoState : BOOL; // the state expected (this test attempts to set the value first);
END_VAR
THIS^.robot := robot;
THIS^.targetDo := targetDo;
THIS^.targetDoState := targetDoState;
END_METHOD

METHOD PRIVATE StateChanged : BOOL
IF  myTestState = prevState THEN
  RETURN;
END_IF

prevState := myTestState;
StateChanged := TRUE;
END_METHOD

METHOD WaitForCycles : BOOL
VAR_INPUT
  maxCount : UINT;
END_VAR
counter := counter + 1;

IF counter = maxCount THEN
  counter := 0;
  WaitForCycles := TRUE;
END_IF
END_METHOD

END_FUNCTION_BLOCK

// ---- Code/RoboConnect/IO Tests/DigitalOutput/T_TcRobot_GetDigitalOutput_IncorrectIndexFails.TcPOU
FUNCTION_BLOCK T_RoboConnect_GetDigitalOutput_IncorrectIndexFails EXTENDS T_UnitTestBase
VAR
  robot : I_RoboConnect;
  targetDO : UINT;
  myTestState, prevState :
    (INIT, ARRANGE, ACT, ASSERT) := INIT;
  expected : BOOL;
  actual : BOOL := TRUE;
  counter : UINT;
  returnedTask : I_Task;
  resultTask : I_BoolResultTask;
END_VAR

CASE myTestState OF
  INIT:
    StateChanged();
    myTestState := ARRANGE;

  ARRANGE:
    IF StateChanged() THEN
      expected := FALSE;
      myTestState := ACT;
    END_IF

  ACT:
    actual := robot.SetDigitalOutput(targetDO, TRUE, task => returnedTask);
    myTestState := ASSERT;

  ASSERT:
    assertion.AssertEquals_BOOL(expected, actual, 'robot.SetDigitalOutput(targetDO, TRUE, task => returnedTask)');
    TestFinished();
    myTestState := INIT;

END_CASE

METHOD FB_init : BOOL
VAR_INPUT
  bInitRetains : BOOL; // if TRUE, the retain variables are initialized (warm start / cold start)
  bInCopyCode : BOOL; // if TRUE, the instance afterwards gets moved into the copy code (online change)
  TestSuite : tcl_SimpleUnitTestLibrary.I_TestSuite;
  robot : I_TcRobot;
  targetDo : UINT;
END_VAR
THIS^.robot := robot;
THIS^.targetDo := targetDo;
END_METHOD

METHOD PRIVATE StateChanged : BOOL
IF  myTestState = prevState THEN
  RETURN;
END_IF

prevState := myTestState;
StateChanged := TRUE;
END_METHOD

METHOD WaitForCycles : BOOL
VAR_INPUT
  maxCount : UINT;
END_VAR
counter := counter + 1;

IF counter = maxCount THEN
  counter := 0;
  WaitForCycles := TRUE;
END_IF
END_METHOD

END_FUNCTION_BLOCK

// ---- Code/RoboConnect/IO Tests/ToolAnalogOutput/T_TcRobot_GetToolAnalogOutput_CorrectIndexPasses.TcPOU
FUNCTION_BLOCK T_RoboConnect_GetToolAnalogOutput_CorrectIndexPasses EXTENDS T_UnitTestBase
VAR
  robot : I_RoboConnect;
  targetDO : UINT;
  myTestState, prevState :
    (INIT, ARRANGE, ACT, ASSERT) := INIT;
  expected, actual : BOOL;
  counter : UINT;
  returnedTask : I_Task;
  resultTask : I_NumberResultTask;
END_VAR

CASE myTestState OF
  INIT:
    StateChanged();
    myTestState := ARRANGE;

  ARRANGE:
    IF StateChanged() THEN
      expected := TRUE;
      myTestState := ACT;
    END_IF

  ACT:
    actual := robot.GetToolAnalogOutput(targetDO, task => resultTask);
    myTestState := ASSERT;

  ASSERT:
    assertion.AssertEquals_BOOL(expected, actual, 'robot.GetToolAnalogOutput(targetDO, task => returnedTask)');
    TestFinished();
    myTestState := INIT;

END_CASE

METHOD FB_init : BOOL
VAR_INPUT
  bInitRetains : BOOL; // if TRUE, the retain variables are initialized (warm start / cold start)
  bInCopyCode : BOOL; // if TRUE, the instance afterwards gets moved into the copy code (online change)
  TestSuite : tcl_SimpleUnitTestLibrary.I_TestSuite;
  robot : I_TcRobot;
  targetDo : UINT;
END_VAR
THIS^.robot := robot;
THIS^.targetDo := targetDo;
END_METHOD

METHOD PRIVATE StateChanged : BOOL
IF  myTestState = prevState THEN
  RETURN;
END_IF

prevState := myTestState;
StateChanged := TRUE;
END_METHOD

METHOD WaitForCycles : BOOL
VAR_INPUT
  maxCount : UINT;
END_VAR
counter := counter + 1;

IF counter = maxCount THEN
  counter := 0;
  WaitForCycles := TRUE;
END_IF
END_METHOD

END_FUNCTION_BLOCK

// ---- Code/RoboConnect/IO Tests/ToolAnalogOutput/T_TcRobot_SetToolAnalogOutput_TimeoutFails.TcPOU
FUNCTION_BLOCK T_RoboConnect_SetToolAnalogOutput_TimeoutFails EXTENDS T_UnitTestBase
VAR
  robot : I_RoboConnect;
  timeOutTimer : TON;
  targetAO : UINT;
  myTestState, prevState :
    (INIT,
    ARRANGE,
    ACT,
    ASSERT) := INIT;
  expected, actual : BOOL;
  counter : UINT;
  returnedTask : I_Task;
END_VAR

CASE myTestState OF
  INIT:
    StateChanged();
    myTestState := ARRANGE;

  ARRANGE:
    IF StateChanged() THEN
      expected := TRUE;
      robot.Connect();
    END_IF

    IF robot.Connected THEN
      myTestState := ACT;
    END_IF

  ACT:
    robot.SetDigitalOutput(targetAO,TRUE, task => returnedTask);
    myTestState := ASSERT;

  ASSERT:
    IF timeOutTimer.Q THEN
      actual := returnedTask.Timeout;
      assertion.AssertEquals_BOOL(expected, actual, 'actual := returnedTask.Timeout');
      TestFinished();
      myTestState := INIT;

    END_IF

END_CASE

robot.CyclicLogic();
timeOutTimer(IN := myTestState = ASSERT);

METHOD FB_init : BOOL
VAR_INPUT
  bInitRetains : BOOL; // if TRUE, the retain variables are initialized (warm start / cold start)
  bInCopyCode : BOOL; // if TRUE, the instance afterwards gets moved into the copy code (online change)
  TestSuite : tcl_SimpleUnitTestLibrary.I_TestSuite;
  robot : I_TcRobot;
  targetAo : UINT;
  timeout : TIME;
END_VAR
THIS^.robot := robot;
THIS^.timeoutTimer.PT := timeout;
THIS^.targetAo := targetAo;
END_METHOD

METHOD PRIVATE StateChanged : BOOL
IF  myTestState = prevState THEN
  RETURN;
END_IF

prevState := myTestState;
StateChanged := TRUE;
END_METHOD

METHOD WaitForCycles : BOOL
VAR_INPUT
  maxCount : UINT;
END_VAR
counter := counter + 1;

IF counter = maxCount THEN
  counter := 0;
  WaitForCycles := TRUE;
END_IF
END_METHOD

END_FUNCTION_BLOCK

// ---- Code/RoboConnect/IO Tests/ToolAnalogOutput/T_TcRobot_SetToolAnalogOutput_IncorrectIndexFails.TcPOU
FUNCTION_BLOCK T_RoboConnect_SetToolAnalogOutput_IncorrectIndexFails EXTENDS T_UnitTestBase
VAR
  robot : I_RoboConnect;
  targetDO : UINT;
  myTestState, prevState :
    (INIT, ARRANGE, ACT, ASSERT)
    := INIT;
  expected : BOOL;
  actual : BOOL := TRUE;
  counter : UINT;
END_VAR

CASE myTestState OF
  INIT:
    StateChanged();
    myTestState := ARRANGE;

  ARRANGE:
    IF StateChanged() THEN
      expected := FALSE;
      myTestState := ACT;
    END_IF

  ACT:
    actual := robot.SetToolAnalogOutput(targetDO, 0.5);
    myTestState := ASSERT;

  ASSERT:
    assertion.AssertEquals_BOOL(expected, actual, 'actual := robot.SetToolAnalogOutput(targetDO, TRUE)');
    TestFinished();
    myTestState := INIT;

END_CASE

METHOD FB_init : BOOL
VAR_INPUT
  bInitRetains : BOOL; // if TRUE, the retain variables are initialized (warm start / cold start)
  bInCopyCode : BOOL; // if TRUE, the instance afterwards gets moved into the copy code (online change)
  TestSuite : tcl_SimpleUnitTestLibrary.I_TestSuite;
  robot : I_TcRobot;
  targetDo : UINT;
END_VAR
THIS^.robot := robot;
THIS^.targetDo := targetDo;
END_METHOD

METHOD PRIVATE StateChanged : BOOL
IF  myTestState = prevState THEN
  RETURN;
END_IF

prevState := myTestState;
StateChanged := TRUE;
END_METHOD

METHOD WaitForCycles : BOOL
VAR_INPUT
  maxCount : UINT;
END_VAR
counter := counter + 1;

IF counter = maxCount THEN
  counter := 0;
  WaitForCycles := TRUE;
END_IF
END_METHOD

END_FUNCTION_BLOCK

// ---- Code/RoboConnect/IO Tests/ToolAnalogOutput/T_TcRobot_SetToolAnalogOutput_CorrectIndexPasses.TcPOU
FUNCTION_BLOCK T_RoboConnect_SetToolAnalogOutput_CorrectIndexPasses EXTENDS T_UnitTestBase
VAR
  robot : I_RoboConnect;
  targetDO : UINT;
  myTestState, prevState :
    (INIT, ARRANGE, ACT, ASSERT) := INIT;
  expected, actual : BOOL;
  counter : UINT;
END_VAR

CASE myTestState OF
  INIT:
    StateChanged();
    myTestState := ARRANGE;

  ARRANGE:
    IF StateChanged() THEN
      expected := TRUE;
      robot.Connect();
    END_IF

    IF robot.Connected THEN
      myTestState := ACT;
    END_IF

  ACT:
    actual := robot.SetToolAnalogOutput(targetDO, 0.5);
    myTestState := ASSERT;

  ASSERT:
    assertion.AssertEquals_BOOL(expected, actual, 'actual := robot.SetToolAnalogOutput(targetDO, TRUE)');
    TestFinished();
    myTestState := INIT;

END_CASE

METHOD FB_init : BOOL
VAR_INPUT
  bInitRetains : BOOL; // if TRUE, the retain variables are initialized (warm start / cold start)
  bInCopyCode : BOOL; // if TRUE, the instance afterwards gets moved into the copy code (online change)
  TestSuite : tcl_SimpleUnitTestLibrary.I_TestSuite;
  robot : I_TcRobot;
  targetDo : UINT;
END_VAR
THIS^.robot := robot;
THIS^.targetDo := targetDo;
END_METHOD

METHOD PRIVATE StateChanged : BOOL
IF  myTestState = prevState THEN
  RETURN;
END_IF

prevState := myTestState;
StateChanged := TRUE;
END_METHOD

METHOD WaitForCycles : BOOL
VAR_INPUT
  maxCount : UINT;
END_VAR
counter := counter + 1;

IF counter = maxCount THEN
  counter := 0;
  WaitForCycles := TRUE;
END_IF
END_METHOD

END_FUNCTION_BLOCK

// ---- Code/RoboConnect/IO Tests/ToolAnalogOutput/T_TcRobot_GetToolAnalogOutput_IncorrectIndexFails.TcPOU
FUNCTION_BLOCK T_RoboConnect_GetToolAnalogOutput_IncorrectIndexFails EXTENDS T_UnitTestBase
VAR
  robot : I_RoboConnect;
  targetDO : UINT;
  myTestState, prevState :
    (INIT,
    ARRANGE,
    ACT,
    ASSERT) := INIT;
  expected : BOOL;
  actual : BOOL := TRUE;
  counter : UINT;
  returnedTask : I_Task;
  resultTask : I_NumberResultTask;
END_VAR

CASE myTestState OF
  INIT:
    StateChanged();
    myTestState := ARRANGE;

  ARRANGE:
    IF StateChanged() THEN
      expected := FALSE;
      myTestState := ACT;
    END_IF

  ACT:
    actual := robot.GetToolAnalogOutput(targetDO, task => resultTask);
    myTestState := ASSERT;

  ASSERT:
    assertion.AssertEquals_BOOL(expected, actual, 'robot.GetToolAnalogOutput(targetDO, task => returnedTask)');
    TestFinished();
    myTestState := INIT;

END_CASE

METHOD FB_init : BOOL
VAR_INPUT
  bInitRetains : BOOL; // if TRUE, the retain variables are initialized (warm start / cold start)
  bInCopyCode : BOOL; // if TRUE, the instance afterwards gets moved into the copy code (online change)
  TestSuite : tcl_SimpleUnitTestLibrary.I_TestSuite;
  robot : I_TcRobot;
  targetDo : UINT;
END_VAR
THIS^.robot := robot;
THIS^.targetDo := targetDo;
END_METHOD

METHOD PRIVATE StateChanged : BOOL
IF  myTestState = prevState THEN
  RETURN;
END_IF

prevState := myTestState;
StateChanged := TRUE;
END_METHOD

METHOD WaitForCycles : BOOL
VAR_INPUT
  maxCount : UINT;
END_VAR
counter := counter + 1;

IF counter = maxCount THEN
  counter := 0;
  WaitForCycles := TRUE;
END_IF
END_METHOD

END_FUNCTION_BLOCK

// ---- Code/RoboConnect/IO Tests/ToolDigitalOutput/T_TcRobot_SetToolDigitalOutputTimeout_Fails.TcPOU
FUNCTION_BLOCK T_RoboConnect_SetToolDigitalOutputTimeout_Fails EXTENDS T_UnitTestBase
VAR
  robot : I_RoboConnect;
  timeOutTimer : TON;
  targetDO : UINT;
  myTestState, prevState :
    (INIT, ARRANGE, ACT, ASSERT) := INIT;
  expected, actual : BOOL;
  counter : UINT;
END_VAR

CASE myTestState OF
  INIT:
    StateChanged();
    myTestState := ARRANGE;

  ARRANGE:
    IF StateChanged() THEN
      expected := TRUE;
      robot.Connect();
    END_IF

    IF robot.Connected THEN
      myTestState := ACT;
    END_IF

  ACT:
    robot.SetToolDigitalOutput(targetDO,TRUE);
    myTestState := ASSERT;

  ASSERT:

    IF timeOutTimer.Q THEN
      actual := robot.GetToolDigitalOutput(targetDO);
      assertion.AssertEquals_BOOL(expected, actual, 'robot.GetDigitalOutput(targetDO) := TRUE');
      TestFinished();
      myTestState := INIT;

    END_IF

END_CASE

timeOutTimer(IN := myTestState = ASSERT);

METHOD FB_init : BOOL
VAR_INPUT
  bInitRetains : BOOL; // if TRUE, the retain variables are initialized (warm start / cold start)
  bInCopyCode : BOOL; // if TRUE, the instance afterwards gets moved into the copy code (online change)
  TestSuite : tcl_SimpleUnitTestLibrary.I_TestSuite;
  robot : I_TcRobot;
  timeout : TIME;
  targetDo : UINT;
END_VAR
THIS^.robot := robot;
THIS^.timeOutTimer.PT := timeout;
THIS^.targetDo := targetDo;
END_METHOD

METHOD PRIVATE StateChanged : BOOL
IF  myTestState = prevState THEN
  RETURN;
END_IF

prevState := myTestState;
StateChanged := TRUE;
END_METHOD

METHOD WaitForCycles : BOOL
VAR_INPUT
  maxCount : UINT;
END_VAR
counter := counter + 1;

IF counter = maxCount THEN
  counter := 0;
  WaitForCycles := TRUE;
END_IF
END_METHOD

END_FUNCTION_BLOCK

// ---- Code/RoboConnect/IO Tests/ToolDigitalOutput/T_TcRobot_GetToolDigitalOutput_CorrectIndexPasses.TcPOU
FUNCTION_BLOCK T_RoboConnect_GetToolDigitalOutput_CorrectIndexPasses EXTENDS T_UnitTestBase
VAR
  robot : I_RoboConnect;
  targetDO : UINT;
  myTestState, prevState :
    (INIT, ARRANGE, ACT, ASSERT) := INIT;
  expected, actual : BOOL;
  counter : UINT;
  returnedTask : I_Task;
  resultTask : I_BoolResultTask;
END_VAR

CASE myTestState OF
  INIT:
    StateChanged();
    myTestState := ARRANGE;

  ARRANGE:
    IF StateChanged() THEN
      expected := TRUE;
      myTestState := ACT;
    END_IF

  ACT:
    actual := robot.GetToolDigitalOutput(targetDO, task => resultTask);
    myTestState := ASSERT;

  ASSERT:
    assertion.AssertEquals_BOOL(expected, actual, 'robot.GetDigitalOutput(targetDO) := TRUE');
    TestFinished();
    myTestState := INIT;

END_CASE

METHOD FB_init : BOOL
VAR_INPUT
  bInitRetains : BOOL; // if TRUE, the retain variables are initialized (warm start / cold start)
  bInCopyCode : BOOL; // if TRUE, the instance afterwards gets moved into the copy code (online change)
  TestSuite : tcl_SimpleUnitTestLibrary.I_TestSuite;
  robot : I_TcRobot;
  targetDo : UINT;
END_VAR
THIS^.robot := robot;
THIS^.targetDo := targetDo;
END_METHOD

METHOD PRIVATE StateChanged : BOOL
IF  myTestState = prevState THEN
  RETURN;
END_IF

prevState := myTestState;
StateChanged := TRUE;
END_METHOD

METHOD WaitForCycles : BOOL
VAR_INPUT
  maxCount : UINT;
END_VAR
counter := counter + 1;

IF counter = maxCount THEN
  counter := 0;
  WaitForCycles := TRUE;
END_IF
END_METHOD

END_FUNCTION_BLOCK

// ---- Code/RoboConnect/IO Tests/ToolDigitalOutput/T_TcRobot_SetToolDigitalOutput_IncorrectIndexFails.TcPOU
FUNCTION_BLOCK T_RoboConnect_SetToolDigitalOutput_IncorrectIndexFails EXTENDS T_UnitTestBase
VAR
  robot : I_RoboConnect;
  targetDO : UINT;
  myTestState, prevState :
    (INIT, ARRANGE, ACT, ASSERT)
    := INIT;
  expected : BOOL;
  actual : BOOL := TRUE;
  counter : UINT;
END_VAR

CASE myTestState OF
  INIT:
    StateChanged();
    myTestState := ARRANGE;

  ARRANGE:
    IF StateChanged() THEN
      expected := FALSE;
      myTestState := ACT;
    END_IF

  ACT:
    actual := robot.SetToolDigitalOutput(targetDO, TRUE);
    myTestState := ASSERT;

  ASSERT:
    assertion.AssertEquals_BOOL(expected, actual, 'robot.GetDigitalOutput(targetDO) := TRUE');
    TestFinished();
    myTestState := INIT;

END_CASE

METHOD FB_init : BOOL
VAR_INPUT
  bInitRetains : BOOL; // if TRUE, the retain variables are initialized (warm start / cold start)
  bInCopyCode : BOOL; // if TRUE, the instance afterwards gets moved into the copy code (online change)
  TestSuite : tcl_SimpleUnitTestLibrary.I_TestSuite;
  robot : I_TcRobot;
  targetDo : UINT;
END_VAR
THIS^.robot := robot;
THIS^.targetDo := targetDo;
END_METHOD

METHOD PRIVATE StateChanged : BOOL
IF  myTestState = prevState THEN
  RETURN;
END_IF

prevState := myTestState;
StateChanged := TRUE;
END_METHOD

METHOD WaitForCycles : BOOL
VAR_INPUT
  maxCount : UINT;
END_VAR
counter := counter + 1;

IF counter = maxCount THEN
  counter := 0;
  WaitForCycles := TRUE;
END_IF
END_METHOD

END_FUNCTION_BLOCK

// ---- Code/RoboConnect/IO Tests/ToolDigitalOutput/T_TcRobot_SetToolDigitalOutput_CorrectIndexPasses.TcPOU
FUNCTION_BLOCK T_RoboConnect_SetToolDigitalOutput_CorrectIndexPasses EXTENDS T_UnitTestBase
VAR
  robot : I_RoboConnect;
  targetDO : UINT;
  myTestState, prevState :
    (INIT, ARRANGE, ACT, ASSERT) := INIT;
  expected, actual : BOOL;
  counter : UINT;
END_VAR

CASE myTestState OF
  INIT:
    StateChanged();
    myTestState := ARRANGE;

  ARRANGE:
    IF StateChanged() THEN
      expected := TRUE;
      myTestState := ACT;
    END_IF

  ACT:
    actual := robot.SetToolDigitalOutput(targetDO, TRUE);
    myTestState := ASSERT;

  ASSERT:
    assertion.AssertEquals_BOOL(expected, actual, 'robot.GetDigitalOutput(targetDO) := TRUE');
    TestFinished();
    myTestState := INIT;

END_CASE

METHOD FB_init : BOOL
VAR_INPUT
  bInitRetains : BOOL; // if TRUE, the retain variables are initialized (warm start / cold start)
  bInCopyCode : BOOL; // if TRUE, the instance afterwards gets moved into the copy code (online change)
  TestSuite : tcl_SimpleUnitTestLibrary.I_TestSuite;
  robot : I_TcRobot;
  targetDo : UINT;
END_VAR
THIS^.robot := robot;
THIS^.targetDo := targetDo;
END_METHOD

METHOD PRIVATE StateChanged : BOOL
IF  myTestState = prevState THEN
  RETURN;
END_IF

prevState := myTestState;
StateChanged := TRUE;
END_METHOD

METHOD WaitForCycles : BOOL
VAR_INPUT
  maxCount : UINT;
END_VAR
counter := counter + 1;

IF counter = maxCount THEN
  counter := 0;
  WaitForCycles := TRUE;
END_IF
END_METHOD

END_FUNCTION_BLOCK

// ---- Code/RoboConnect/IO Tests/ToolDigitalOutput/T_TcRobot_GetToolDigitalOutput_IncorrectIndexFails.TcPOU
FUNCTION_BLOCK T_RoboConnect_GetToolDigitalOutput_IncorrectIndexFails EXTENDS T_UnitTestBase
VAR
  robot : I_RoboConnect;
  targetDO : UINT;
  myTestState, prevState :
    (INIT,
    ARRANGE,
    ACT,
    ASSERT) := INIT;
  expected : BOOL;
  actual : BOOL := TRUE;
  counter : UINT;
  returnedTask : I_Task;
  resultTask : I_BoolResultTask;
END_VAR

CASE myTestState OF
  INIT:
    StateChanged();
    myTestState := ARRANGE;

  ARRANGE:
    IF StateChanged() THEN
      expected := FALSE;
      myTestState := ACT;
    END_IF

  ACT:
    actual := robot.GetToolDigitalOutput(targetDO, task => resultTask);
    myTestState := ASSERT;

  ASSERT:
    assertion.AssertEquals_BOOL(expected, actual, 'robot.GetToolDigitalOutput(targetDO, task => returnedTask)');
    TestFinished();
    myTestState := INIT;

END_CASE

METHOD FB_init : BOOL
VAR_INPUT
  bInitRetains : BOOL; // if TRUE, the retain variables are initialized (warm start / cold start)
  bInCopyCode : BOOL; // if TRUE, the instance afterwards gets moved into the copy code (online change)
  TestSuite : tcl_SimpleUnitTestLibrary.I_TestSuite;
  robot : I_TcRobot;
  targetDo : UINT;
END_VAR
THIS^.robot := robot;
THIS^.targetDo := targetDo;
END_METHOD

METHOD PRIVATE StateChanged : BOOL
IF  myTestState = prevState THEN
  RETURN;
END_IF

prevState := myTestState;
StateChanged := TRUE;
END_METHOD

METHOD WaitForCycles : BOOL
VAR_INPUT
  maxCount : UINT;
END_VAR
counter := counter + 1;

IF counter = maxCount THEN
  counter := 0;
  WaitForCycles := TRUE;
END_IF
END_METHOD

END_FUNCTION_BLOCK

// ---- Code/RoboConnect/IO Tests/ToolDigitalOutput/T_TcRobot_SetToolDigitalOutput_ReturnsTrueOutput.TcPOU
FUNCTION_BLOCK T_RoboConnect_SetToolDigitalOutput_ReturnsTrueOutput EXTENDS T_UnitTestBase
VAR
  robot : I_RoboConnect;
  timeOutTimer : TON;
  targetDO : UINT;
  myTestState, prevState :
    (INIT,
    ARRANGE,
    ACT,
    ASSERT) := INIT;
  expected, actual : BOOL;
  counter : UINT;
  returnedTask : I_Task;
  resultTask : I_BoolResultTask;
END_VAR

CASE myTestState OF
  INIT:
    StateChanged();
    myTestState := ARRANGE;

  ARRANGE:
    IF StateChanged() THEN
      expected := TRUE;
      robot.Connect();
    END_IF

    IF robot.Connected THEN
      myTestState := ACT;
    END_IF

  ACT:
    robot.SetToolDigitalOutput(targetDO, TRUE, task => returnedTask);
    myTestState := ASSERT;

  ASSERT:

    IF timeOutTimer.Q THEN
      actual := robot.GetToolDigitalOutput(targetDO, task => resultTask);
      assertion.AssertEquals_BOOL(expected, actual, 'actual := robot.GetToolDigitalOutput(targetDO, task => resultTask)');
      TestFinished();
      myTestState := INIT;

    END_IF

END_CASE

timeOutTimer(IN := myTestState = ASSERT);

METHOD FB_init : BOOL
VAR_INPUT
  bInitRetains : BOOL; // if TRUE, the retain variables are initialized (warm start / cold start)
  bInCopyCode : BOOL; // if TRUE, the instance afterwards gets moved into the copy code (online change)
  TestSuite : tcl_SimpleUnitTestLibrary.I_TestSuite;
  robot : I_TcRobot;
  timeout : TIME;
  targetDo : UINT;
END_VAR
THIS^.robot := robot;
THIS^.timeOutTimer.PT := timeout;
THIS^.targetDo := targetDo;
END_METHOD

METHOD PRIVATE StateChanged : BOOL
IF  myTestState = prevState THEN
  RETURN;
END_IF

prevState := myTestState;
StateChanged := TRUE;
END_METHOD

METHOD WaitForCycles : BOOL
VAR_INPUT
  maxCount : UINT;
END_VAR
counter := counter + 1;

IF counter = maxCount THEN
  counter := 0;
  WaitForCycles := TRUE;
END_IF
END_METHOD

END_FUNCTION_BLOCK

// ---- Code/RoboConnect/T_TcRobot_DisableNotConnected_ReturnsFalse.TcPOU
FUNCTION_BLOCK T_RoboConnect_DisableNotConnected_ReturnsFalse EXTENDS T_UnitTestBase
VAR
  robot : T_MockRoboConnect;
  expected : BOOL := FALSE;
  actual : BOOL := TRUE;
END_VAR

actual := robot.Disable();
assertion.AssertEquals_BOOL(expected, actual, 'actual := robot.Disable();');
TestFinished();

END_FUNCTION_BLOCK

// ---- Code/RoboConnect/T_TcRobot_MoveJWrongCount_ReturnsFalse.TcPOU
FUNCTION_BLOCK T_RoboConnect_MoveJWrongCount_ReturnsFalse EXTENDS T_UnitTestBase
VAR
  robot : T_MockRoboConnect;
  targets : ARRAY [1..4] OF LREAL;
  expected : BOOL := FALSE;
  actual : BOOL := TRUE;
END_VAR

actual := robot.MoveJ(targets);
assertion.AssertEquals_BOOL(expected, actual, 'actual := robot.MoveJ(targets)');
TestFinished();

END_FUNCTION_BLOCK
